TYPE HMI_ERR_TemplateMachinePart :
STRUCT
	(*
		Rules:
		Errors shall only be off type BOOL
		Errors shall be set >> the HMI block will do the resetting

		Syntax convention:
		a clear variable name which describes the error			as described below
		InitNotEmpty:BOOL;										//Error [machinepart]: not empty during initialisation
		
		prio's: emergency stop items == 100, e-circuit=99, default (nothing specified) = 50
		adjust as needed
		//example how to pre-set error priorities for the HMI. Default errors get prio 50, Recommend prio 100 for e-stop buttons etc
		ExampleAddPrioForHmiError:BOOL;					//Error[prio=90] TemplateMachinePart: we have an error!
	*)
	InitNotEmpty:BOOL;								//Error [machinepart]: not empty during initialisation
	
	//example how to pre-set error priorities for the HMI. Default errors get prio 50, Recommend prio 100 for e-stop buttons etc
	ExampleAddPrioForHmiError:BOOL;					//Error[prio=100] TemplateMachinePart: we have an error!
	
	//test log error by name, very long name, truncation
	TestStupidLongErrorNameWillItGetLoggedAbcdefghijklmnopqrstuvwzyzAbcdefghijklmnopqrstuvwzyzAbcdefghijklmnopqrstuvwzyzAbcdefghijklmnopqrstuvwzyzAbcdefghijklmnopqrstuvwzyz:BOOL;
END_STRUCT
END_TYPE

(* stored: Version 1.1.0.1
   DUT HMI_ERR_TemplateMachinePart: Id {c179f755-97ec-450e-b3c8-480ebcff4cb9} *)
